TYPE URL :
STRUCT
	PROTOCOL : STRING(10);
	USER : STRING(32);
	PASSWORD : STRING(32);
	DOMAIN : STRING(80);
	PORT : WORD;
	PATH : STRING(80);
	QUERY : STRING(STRING_LENGTH);
	ANCHOR : STRING(40);
	HEADER : STRING(160);
END_STRUCT
END_TYPE

(* stored: Version 1.1.0.1, ProductVersion 3.1.4024.4
   DUT URL: Id {1e48f2fa-6fc5-4661-bf39-995115c3015e} *)
